{attribute 'linkalways'} 
{attribute 'no_explicit_call' := 'This FB is a CLASS and must be accessed using methods or properties'}
{attribute 'enable_dynamic_creation'}
FUNCTION_BLOCK FINAL Node_XOR EXTENDS Node
VAR
	in1 : _BOOL(FALSE);
    in2 : _BOOL(FALSE);
	out : _BOOL(FALSE);
END_VAR

METHOD PUBLIC  Clone : I_Node
VAR
	pNode : POINTER TO Node_XOR;
END_VAR
pNode := __NEW(Node_XOR);
Clone := pNode^;
END_METHOD

METHOD FB_init : BOOL
VAR_INPUT
	bInitRetains : BOOL; // if TRUE, the retain variables are initialized (warm start / cold start)
	bInCopyCode : BOOL;  // if TRUE, the instance afterwards gets moved into the copy code (online change)
END_VAR
AddParameter('in1', in1);
AddParameter('in2', in2);
AddOutput('out', out);

this^.Metadatum.AddBoolAsMetadata('deprecated', true);
END_METHOD

METHOD PROTECTED OnExecute
VAR
END_VAR
out.Value := in1.Value XOR in2.Value;
END_METHOD

END_FUNCTION_BLOCK

(* stored: Version 1.1.0.1, ProductVersion 3.1.4026.18
   POU Node_XOR: Id {8188f083-6946-0dd8-1732-4ffeb201ad79}, SpecialFunc None
   Folder Constructor: Id {bff134f8-9c03-0340-0214-c003614c74d3}
   Method Clone: Id {467a3cfb-faff-0004-0bf4-930e1ae4e4ff}
   Method FB_init: Id {3a174d49-40f6-03d6-25ee-8c4371eff331}
   Method OnExecute: Id {562d82c3-1c8f-0cdc-3331-57d495103da6} *)
